FUNCTION_BLOCK EventWrapper3 (* Composite Function Block Type *)
  (* Standard: 61499-2 *)
  (* Version 0.0, 4/9/2019, erik, nxtControl GmbH, template *)
  PACKAGE Main;
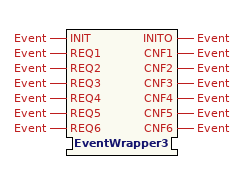
  EVENT_INPUT
    INIT; (* Initialization Request *)
    REQ1; (* Normal Execution Request *)
    REQ2;
    REQ3;
    REQ4;
    REQ5;
    REQ6;
  END_EVENT
  EVENT_OUTPUT
    INITO; (* Initialization Confirm *)
    CNF1; (* Execution Confirmation *)
    CNF2;
    CNF3;
    CNF4;
    CNF5;
    CNF6;
  END_EVENT
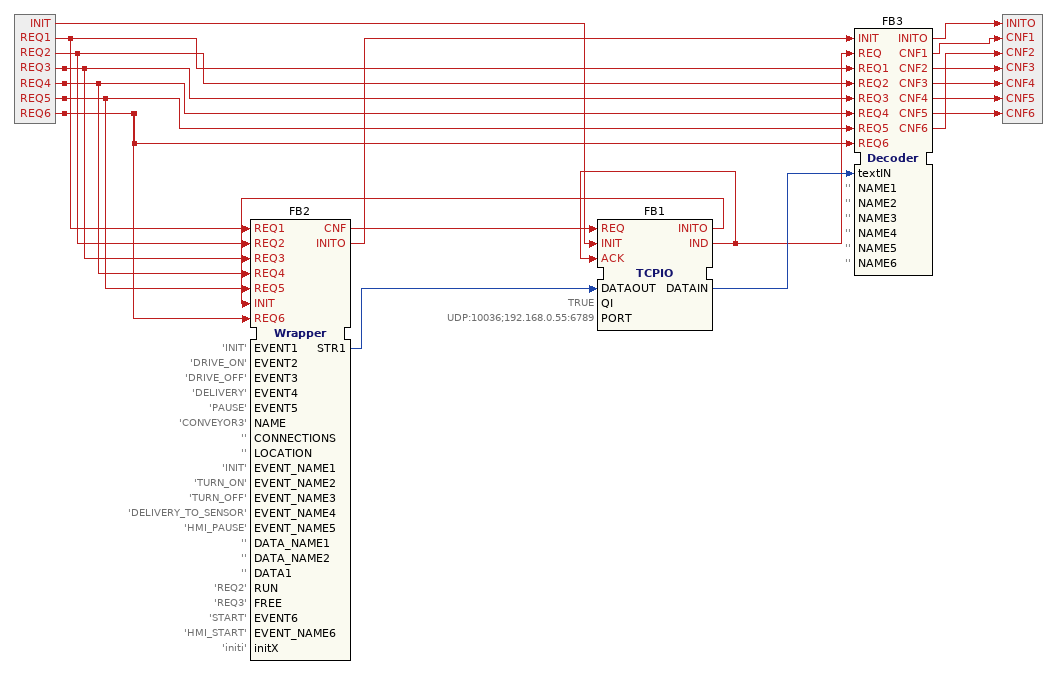
  FBS
    FB1 : TCPIO(QI := TRUE, PORT := UDP:10036;192.168.0.55:6789);
    FB2 : Wrapper(EVENT1 := 'INIT', EVENT2 := 'DRIVE_ON', EVENT3 := 'DRIVE_OFF', EVENT4 := 'DELIVERY', EVENT5 := 'PAUSE', NAME := 'CONVEYOR3', CONNECTIONS := '', LOCATION := '', EVENT_NAME1 := 'INIT', EVENT_NAME2 := 'TURN_ON', EVENT_NAME3 := 'TURN_OFF', EVENT_NAME4 := 'DELIVERY_TO_SENSOR', EVENT_NAME5 := 'HMI_PAUSE', DATA_NAME1 := '', DATA_NAME2 := '', DATA1 := '', RUN := 'REQ2', FREE := 'REQ3', EVENT6 := 'START', EVENT_NAME6 := 'HMI_START', initX := 'initi');
    FB3 : Decoder(NAME1 := '', NAME2 := '', NAME3 := '', NAME4 := '', NAME5 := '', NAME6 := '');
  END_FBS
  EVENT_CONNECTIONS
    REQ1 TO FB2.REQ1;
    REQ2 TO FB2.REQ2;
    REQ3 TO FB2.REQ3;
    FB2.CNF TO FB1.REQ;
    REQ4 TO FB2.REQ4;
    REQ5 TO FB2.REQ5;
    INIT TO FB1.INIT;
    FB1.INITO TO FB2.INIT;
    FB1.IND TO FB1.ACK;
    REQ6 TO FB2.REQ6;
    FB1.IND TO FB3.REQ;
    FB3.INITO TO INITO;
    FB3.CNF3 TO CNF3;
    FB3.CNF2 TO CNF2;
    FB3.CNF1 TO CNF1;
    FB3.CNF4 TO CNF4;
    FB3.CNF5 TO CNF5;
    FB3.CNF6 TO CNF6;
    REQ1 TO FB3.REQ1;
    REQ2 TO FB3.REQ2;
    REQ3 TO FB3.REQ3;
    REQ4 TO FB3.REQ4;
    REQ5 TO FB3.REQ5;
    REQ6 TO FB3.REQ6;
    FB2.INITO TO FB3.INIT;
  END_CONNECTIONS
  DATA_CONNECTIONS
    FB2.STR1 TO FB1.DATAOUT;
    FB1.DATAIN TO FB3.textIN;
  END_CONNECTIONS
END_FUNCTION_BLOCK
